// Brief: Slave Arm Gravity Calibration
FUNCTION_BLOCK PUBLIC FB_SlaveCtrlGraCali EXTENDS FB_SlaveArmCtrlBase
VAR_INPUT
END_VAR
VAR_OUTPUT
END_VAR
VAR
// cali trajectory
	m_caliMotionSegs :INT :=3;
	m_graCaliTraj:ARRAY [1..3, 1..g_sJntNum] OF LREAL:=
		[-pi/6, -PI/2+pi/6, 0.5, 	5(-pi/3),
		 pi/6, 	-PI/2-pi/4, 0.3, 	5(0),
		 -pi/6, -PI/2+pi/6, 0.5, 	5(-pi/3)];
		 
	m_caliMaxjntVel:Vec8d:=[2(2.5*g_deg2Rad), 0.01, 5(2.5*g_deg2Rad)];
	m_caliMaxjntAcc:Vec8d:=[8(0.5)];
	m_caliMaxjntJerk:Vec8d:=[8(2.0)];
	
	m_caliTrajIdx: INT := 1;
	m_caliPlanner: ARRAY[1..3] OF FB_TrajMoveJ;
	
END_VAR

// override this function in each exact controller
METHOD PROTECTED calcCmdJntPos : BOOL
VAR_IN_OUT CONSTANT
	i_endoscopePose : ST_Frame;
	i_masterStatus :ST_MasterStatus;
	i_setupStatus: ST_SetupStatus;
	i_slaveArm :FB_SlaveArm;
END_VAR


VAR 
	i :INT;
	curJntVel :Vec8d;
END_VAR
// check if planner is ready
IF m_caliPlanner[m_caliTrajIdx].isGene = FALSE THEN
	calcCmdJntPos:=FALSE;
	RETURN;
END_IF

// traj plan
calcCmdJntPos :=m_caliPlanner[m_caliTrajIdx].evaluate(m_timePeriod, jntPos=> m_cmdJntPos, jntVel=>m_cmdJntVel, jntAcc=> m_cmdJntAcc);

// check if to transit to next segment
curJntVel :=i_slaveArm.curJntVel;
IF(m_timePeriod > m_caliPlanner[m_caliTrajIdx].duration  AND norm(curJntVel)<7*GVL_SlaveControlParameters.g_jntStaticVelThres) THEN
	m_caliTrajIdx:=m_caliTrajIdx+1;
	m_timePeriod:=0;
END_IF

// check if to terminated
IF(m_caliTrajIdx > m_caliMotionSegs) THEN
	m_isFinished:=TRUE;
END_IF
END_METHOD

METHOD PUBLIC init : BOOL
VAR_IN_OUT CONSTANT
	i_slaveArm	:FB_SlaveArm;
END_VAR
VAR_IN_OUT 
	r_slaveArmCtrlCmd :ST_SlaveArmCtrlCmds;
END_VAR

VAR
	i,j :INT;
	initJntPos,startJntPos,endJntPos :Vec8d;

END_VAR
SUPER^.Init(i_slaveArm,r_slaveArmCtrlCmd);
m_caliTrajIdx :=1;
m_jntOPMode := g_slaveAllPosTrqMode;

// traj plan
// fisrt segment
initJntPos:=i_slaveArm.curJntPos;
startJntPos:=initJntPos;
endJntPos:=startJntPos;
FOR j:=1 TO g_sJntNum DO 
	IF j>3 THEN
		endJntPos[j]:=initJntPos[j]+ m_graCaliTraj[1,j];
	ELSE
		endJntPos[j]:=m_graCaliTraj[1,j];
	END_IF
END_FOR
m_caliPlanner[1].init(startJntPos,endJntPos,m_caliMaxjntVel, m_caliMaxJntAcc, m_caliMaxJntJerk);

// other segments
FOR i:=2 TO m_caliMotionSegs DO 
	startJntPos := endJntPos;
	FOR j:=1 TO g_sJntNum DO 
		IF j>3 THEN
			endJntPos[j]:=initJntPos[j]+ m_graCaliTraj[i,j];
		ELSE
			endJntPos[j]:=m_graCaliTraj[i,j];
		END_IF
	END_FOR
	m_caliPlanner[i].init(startJntPos,endJntPos,m_caliMaxjntVel, m_caliMaxJntAcc, m_caliMaxJntJerk);
END_FOR

// update commands to arm
copyCmds(r_slaveArmCtrlCmd);
END_METHOD

END_FUNCTION_BLOCK

(* stored: Version 1.1.0.1, ProductVersion 3.1.4024.11
   POU FB_SlaveCtrlGraCali: Id {9ec40fb0-5513-4ed9-babf-e07e71772a70}, SpecialFunc None
   Method calcCmdJntPos: Id {e8388ef5-ff5f-4bc0-805c-b4f37a5ed6ad}
   Method init: Id {1fed4a27-3de6-4ef1-8a15-2cb2fd5aafb3} *)
